FUNCTION_BLOCK VCylAdp (* Composite Function Block Type *)
  (* Standard: 61499-2 *)
  (* Version 0.0, 06/10/2018, Atmojo, nxtControl GmbH, template *)
  PACKAGE Main;
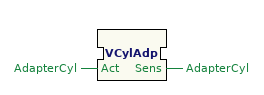
  SOCKETS
    Act : AdapterCyl;
  END_SOCKETS
  PLUGS
    Sens : AdapterCyl;
  END_PLUGS
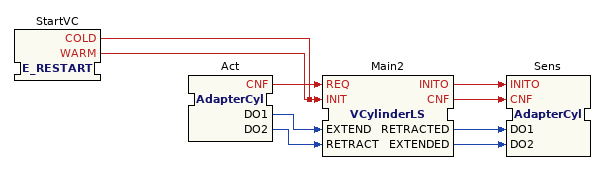
  FBS
    Main2 : VCylinderLS;
    StartVC : E_RESTART;
  END_FBS
  EVENT_CONNECTIONS
    Main2.INITO TO Sens.INITO;
    Act.CNF TO Main2.REQ;
    Main2.CNF TO Sens.CNF;
    StartVC.COLD TO Main2.INIT;
    StartVC.WARM TO Main2.INIT;
  END_CONNECTIONS
  DATA_CONNECTIONS
    Act.DO1 TO Main2.EXTEND;
    Act.DO2 TO Main2.RETRACT;
    Main2.RETRACTED TO Sens.DO1;
    Main2.EXTENDED TO Sens.DO2;
  END_CONNECTIONS
END_FUNCTION_BLOCK
